TYPE ST_AirPressureParCmd :
STRUCT
    Reserved : BOOL; // passive monitor: physical four-structure contract, no command payload
END_STRUCT
END_TYPE

(* stored: Version 1.1.0.1, ProductVersion 3.1.4024.12
   DUT ST_AirPressureParCmd: Id {a37ce1e3-4e13-4009-b607-af4c7df9162a} *)
